// TIA Portal V15 export
// export: Created 2018-05-30T14:06:10.2711692Z, ExportSetting WithDefaults, WithReadOnly, DisplayName Totally Integrated Automation Portal, DisplayVersion V15, DisplayName TIA Portal Openness, DisplayVersion V15, DisplayName STEP 7 Professional, DisplayVersion V15, DisplayName WinCC Professional, DisplayVersion V15
FUNCTION_BLOCK "BST_SINAG120_400"   // FB22, STL
{ S7_Optimized_Access := 'FALSE' }
VERSION : 0.1
// stored: AutoNumber false, CodeModifiedDate 2018-05-30T14:00:08.4304732Z, CompileDate 2018-05-30T14:00:08.4304731Z, CreationDate 2018-05-30T13:56:31.6980767Z, InterfaceModifiedDate 2018-05-30T13:59:44.6951155Z, IsConsistent true, IsKnowHowProtected false, ISMultiInstanceCapable true, IsWriteProtected false, LibraryConformanceStatus The object is library-conformant., ModifiedDate 2018-05-30T14:00:08.4304732Z, ParameterModified 2018-05-30T13:59:44.6951155Z, StructureModified 2018-05-30T13:59:44.6951155Z, UDAEnableTagReadback false
   VAR_INPUT
      L_ON : Bool;
      L_AUT : Bool;
   END_VAR
   VAR_OUTPUT
      QNOFF2 : Bool;
      QERR : Bool;
      QERR_EXT : Bool;
   END_VAR
BEGIN
END_FUNCTION_BLOCK
